// TIA Portal project "Project3" (V17)

(* hardware
DEVICE "S7-1200 station_1"  S7-1200 Station
   slot 0: "Rack_0"  S7-1200 Rack  Rack  V1.0
   slot 1: "PLC_1"  CPU 1214C AC/DC/Rly  6ES7 214-1BG40-0XB0  V4.2
*)

// ===== PLC "PLC_1"  CPU 1214C AC/DC/Rly =====

VAR_GLOBAL   // PLC tag table "Default tag table"
   "PB0" AT %I0.0 : Bool;
   "PB1" AT %I0.1 : Bool;
   "PB2" AT %I0.2 : Bool;
   "PL1" AT %Q0.0 : Bool;
   "PL2" AT %Q0.1 : Bool;
   "X1" AT %M0.0 : Bool;
   "X2" AT %M0.1 : Bool;
END_VAR

ORGANIZATION_BLOCK "Main"   // OB1, LAD, ProgramCycle
TITLE = "Main Program Sweep (Cycle)"
{ S7_Optimized_Access := 'TRUE' }
VERSION : 0.1
   VAR_INPUT
      Initial_Call : Bool;   // Initial call of this OB
      Remanence : Bool;   // =True, if remanent data are available
   END_VAR
BEGIN

REGION Network 1
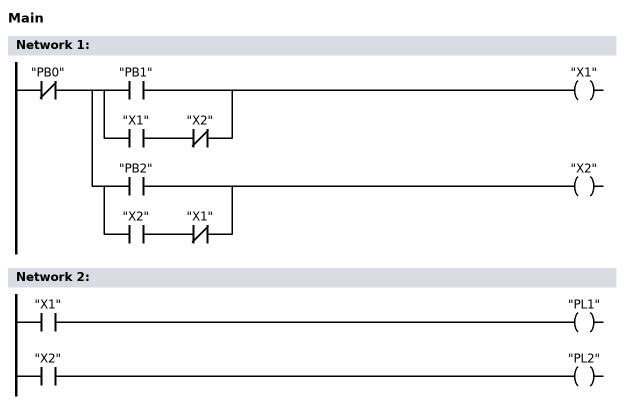
   RUNG wire#powerrail
      I_Contact( "PB0" )
      wire#w1
      Contact( "PB1" )
      wire#w2
      Coil( "X1" )
   END_RUNG
   RUNG wire#w1
      Contact( "X1" )
      I_Contact( "X2" )
   END_RUNG wire#w2
   RUNG wire#w1
      Contact( "PB2" )
      wire#w3
      Coil( "X2" )
   END_RUNG
   RUNG wire#w1
      Contact( "X2" )
      I_Contact( "X1" )
   END_RUNG wire#w3
   // the same network as SCL:
   "X1" := NOT "PB0" AND ("PB1" OR ("X1" AND NOT "X2"));
   "X2" := NOT "PB0" AND ("PB2" OR ("X2" AND NOT "X1"));
END_REGION

REGION Network 2
   RUNG wire#powerrail
      Contact( "X1" )
      Coil( "PL1" )
   END_RUNG
   RUNG wire#powerrail
      Contact( "X2" )
      Coil( "PL2" )
   END_RUNG
   // the same network as SCL:
   "PL1" := "X1";
   "PL2" := "X2";
END_REGION
END_ORGANIZATION_BLOCK